PROGRAM MAIN
VAR
	fbLogger 		: FB_Logger('File.csv');
	retMsg			: STRING;
END_VAR

retMsg := fbLogger.Write('Hello');

END_PROGRAM

(* stored: Version 1.1.0.1, ProductVersion 3.1.0.24
   POU MAIN: Id {fd6e49ae-9c60-4ba4-ba01-45f20a4b6c2c} *)
